// TIA Portal V19 export
FUNCTION_BLOCK "F_Zone29_FB"   // FB168, F_LAD
TITLE = SAFETY ZONE 29 - AREA 03 (SCARICO NAVETTA)
// stored: Access Published
   VAR
      D22_LightCurtain_Ext : "Door_FB";
      D24_LightCurtain_Int : "Door_FB";
      FNS : "ForceNormalStop";
      F_Sinamics_Navetta_Testa : "FDevice_Sinamics_FB";
      F_Sinamics_Navetta_Coda : "FDevice_Sinamics_FB";
      F_SafetyValve_Air_A0304 : "FDevice_Valve_FB";
   END_VAR
   VAR_TEMP
      DoorNormalStop : Bool;
      DoorSafeStop : Bool;
      Door_OK : Bool;
      FDBK : Bool;
   END_VAR
BEGIN

REGION Network 1: < < < < < < < < < < DOOR > > > > > > > > > >
END_REGION

REGION Network 2: Zone Entry enable
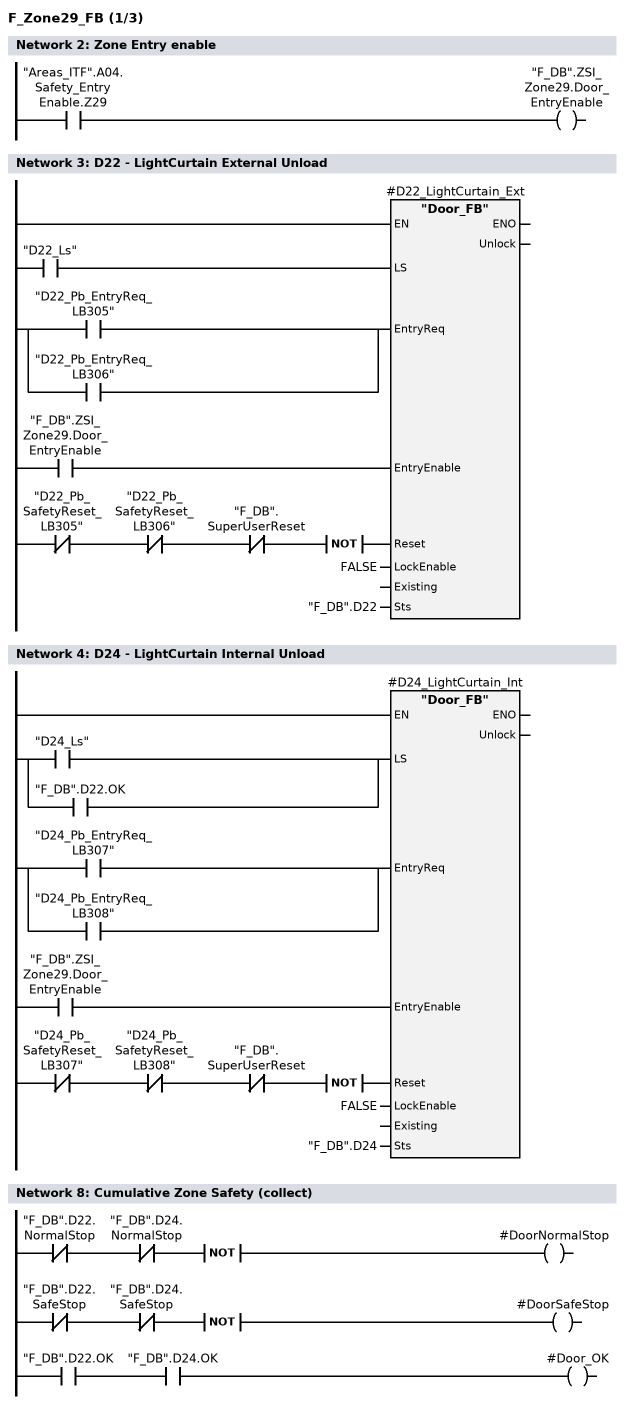
   RUNG wire#powerrail
      Contact( "Areas_ITF".A04.Safety_EntryEnable.Z29 )
      Coil( "F_DB".ZSI_Zone29.Door_EntryEnable )
   END_RUNG
   // the same network as SCL:
   "F_DB".ZSI_Zone29.Door_EntryEnable := "Areas_ITF".A04.Safety_EntryEnable.Z29;
END_REGION

REGION Network 3: D22 - LightCurtain External Unload
   RUNG wire#powerrail
      #D22_LightCurtain_Ext(LS := wire#w1, EntryReq := wire#w2, EntryEnable := wire#w3, Reset := wire#w4, LockEnable := FALSE, Existing :=, Sts := "F_DB".D22, Unlock =>)
   END_RUNG
   RUNG wire#powerrail
      Contact( "D22_Ls" )
   END_RUNG wire#w1
   RUNG wire#powerrail
      Contact( "D22_Pb_EntryReq_LB305" )
   END_RUNG wire#w2
   RUNG wire#powerrail
      Contact( "D22_Pb_EntryReq_LB306" )
   END_RUNG wire#w2
   RUNG wire#powerrail
      Contact( "F_DB".ZSI_Zone29.Door_EntryEnable )
   END_RUNG wire#w3
   RUNG wire#powerrail
      I_Contact( "D22_Pb_SafetyReset_LB305" )
      I_Contact( "D22_Pb_SafetyReset_LB306" )
      I_Contact( "F_DB".SuperUserReset )
      Not()
   END_RUNG wire#w4
   // the same network as SCL:
   #D22_LightCurtain_Ext(LS := "D22_Ls",   // "Door_FB"
                         EntryReq := "D22_Pb_EntryReq_LB305" OR "D22_Pb_EntryReq_LB306",
                         EntryEnable := "F_DB".ZSI_Zone29.Door_EntryEnable,
                         Reset := NOT (NOT "D22_Pb_SafetyReset_LB305" AND NOT "D22_Pb_SafetyReset_LB306" AND NOT "F_DB".SuperUserReset),
                         LockEnable := FALSE,
                         Sts := "F_DB".D22);
END_REGION

REGION Network 4: D24 - LightCurtain Internal Unload
   RUNG wire#powerrail
      #D24_LightCurtain_Int(LS := wire#w1, EntryReq := wire#w2, EntryEnable := wire#w3, Reset := wire#w4, LockEnable := FALSE, Existing :=, Sts := "F_DB".D24, Unlock =>)
   END_RUNG
   RUNG wire#powerrail
      Contact( "D24_Ls" )
   END_RUNG wire#w1
   RUNG wire#powerrail
      Contact( "F_DB".D22.OK )
   END_RUNG wire#w1
   RUNG wire#powerrail
      Contact( "D24_Pb_EntryReq_LB307" )
   END_RUNG wire#w2
   RUNG wire#powerrail
      Contact( "D24_Pb_EntryReq_LB308" )
   END_RUNG wire#w2
   RUNG wire#powerrail
      Contact( "F_DB".ZSI_Zone29.Door_EntryEnable )
   END_RUNG wire#w3
   RUNG wire#powerrail
      I_Contact( "D24_Pb_SafetyReset_LB307" )
      I_Contact( "D24_Pb_SafetyReset_LB308" )
      I_Contact( "F_DB".SuperUserReset )
      Not()
   END_RUNG wire#w4
   // the same network as SCL:
   #D24_LightCurtain_Int(LS := "D24_Ls" OR "F_DB".D22.OK,   // "Door_FB"
                         EntryReq := "D24_Pb_EntryReq_LB307" OR "D24_Pb_EntryReq_LB308",
                         EntryEnable := "F_DB".ZSI_Zone29.Door_EntryEnable,
                         Reset := NOT (NOT "D24_Pb_SafetyReset_LB307" AND NOT "D24_Pb_SafetyReset_LB308" AND NOT "F_DB".SuperUserReset),
                         LockEnable := FALSE,
                         Sts := "F_DB".D24);
END_REGION

REGION Network 7: < < < < < < < < < < ZONE SAFETY INTERFACE > > > > > > > > > >
END_REGION

REGION Network 8: Cumulative Zone Safety (collect)
   RUNG wire#powerrail
      I_Contact( "F_DB".D22.NormalStop )
      I_Contact( "F_DB".D24.NormalStop )
      Not()
      Coil( #DoorNormalStop )
   END_RUNG
   RUNG wire#powerrail
      I_Contact( "F_DB".D22.SafeStop )
      I_Contact( "F_DB".D24.SafeStop )
      Not()
      Coil( #DoorSafeStop )
   END_RUNG
   RUNG wire#powerrail
      Contact( "F_DB".D22.OK )
      Contact( "F_DB".D24.OK )
      Coil( #Door_OK )
   END_RUNG
   // the same network as SCL:
   #DoorNormalStop := NOT (NOT "F_DB".D22.NormalStop AND NOT "F_DB".D24.NormalStop);
   #DoorSafeStop := NOT (NOT "F_DB".D22.SafeStop AND NOT "F_DB".D24.SafeStop);
   #Door_OK := "F_DB".D22.OK AND "F_DB".D24.OK;
END_REGION

REGION Network 9: Zone must stay in Normal Stop During Restart
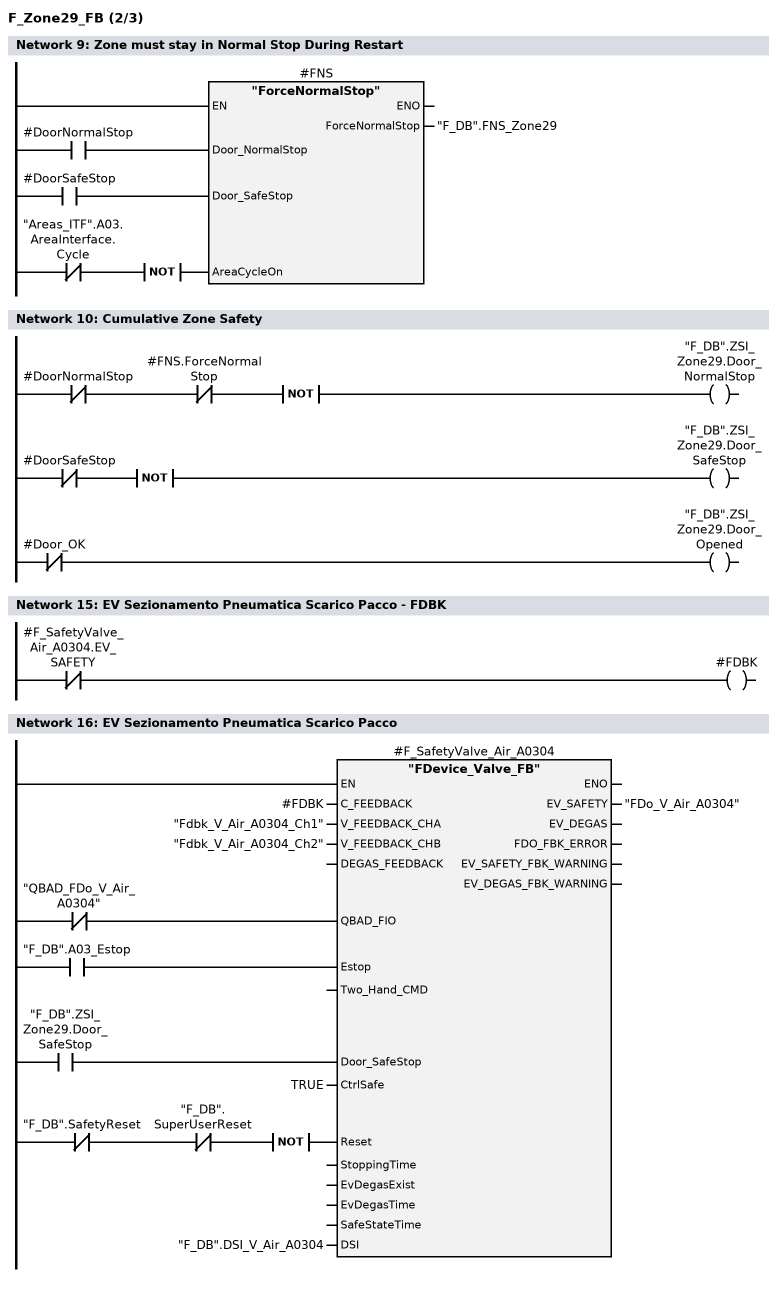
   RUNG wire#powerrail
      #FNS(Door_NormalStop := wire#w1, Door_SafeStop := wire#w2, AreaCycleOn := wire#w3, ForceNormalStop => "F_DB".FNS_Zone29)
   END_RUNG
   RUNG wire#powerrail
      Contact( #DoorNormalStop )
   END_RUNG wire#w1
   RUNG wire#powerrail
      Contact( #DoorSafeStop )
   END_RUNG wire#w2
   RUNG wire#powerrail
      I_Contact( "Areas_ITF".A03.AreaInterface.Cycle )
      Not()
   END_RUNG wire#w3
   // the same network as SCL:
   #FNS(Door_NormalStop := #DoorNormalStop,   // "ForceNormalStop"
        Door_SafeStop := #DoorSafeStop,
        AreaCycleOn := NOT (NOT "Areas_ITF".A03.AreaInterface.Cycle),
        ForceNormalStop => "F_DB".FNS_Zone29);
END_REGION

REGION Network 10: Cumulative Zone Safety
   RUNG wire#powerrail
      I_Contact( #DoorNormalStop )
      I_Contact( #FNS.ForceNormalStop )
      Not()
      Coil( "F_DB".ZSI_Zone29.Door_NormalStop )
   END_RUNG
   RUNG wire#powerrail
      I_Contact( #DoorSafeStop )
      Not()
      Coil( "F_DB".ZSI_Zone29.Door_SafeStop )
   END_RUNG
   RUNG wire#powerrail
      I_Contact( #Door_OK )
      Coil( "F_DB".ZSI_Zone29.Door_Opened )
   END_RUNG
   // the same network as SCL:
   "F_DB".ZSI_Zone29.Door_NormalStop := NOT (NOT #DoorNormalStop AND NOT #FNS.ForceNormalStop);
   "F_DB".ZSI_Zone29.Door_SafeStop := NOT (NOT #DoorSafeStop);
   "F_DB".ZSI_Zone29.Door_Opened := NOT #Door_OK;
END_REGION

REGION Network 11: >
END_REGION

REGION Network 12: >
END_REGION

REGION Network 13: < < < < < < < < < < DEVICES SAFETY VALVES > > > > > > > > > >
END_REGION

REGION Network 14: >
END_REGION

REGION Network 15: EV Sezionamento Pneumatica Scarico Pacco - FDBK
   RUNG wire#powerrail
      I_Contact( #F_SafetyValve_Air_A0304.EV_SAFETY )
      Coil( #FDBK )
   END_RUNG
   // the same network as SCL:
   #FDBK := NOT #F_SafetyValve_Air_A0304.EV_SAFETY;
END_REGION

REGION Network 16: EV Sezionamento Pneumatica Scarico Pacco
   RUNG wire#powerrail
      #F_SafetyValve_Air_A0304(QBAD_FIO := wire#w1, Estop := wire#w2, Door_SafeStop := wire#w3, Reset := wire#w4, C_FEEDBACK := #FDBK, V_FEEDBACK_CHA := "Fdbk_V_Air_A0304_Ch1", V_FEEDBACK_CHB := "Fdbk_V_Air_A0304_Ch2", DEGAS_FEEDBACK :=, Two_Hand_CMD :=, CtrlSafe := TRUE, StoppingTime :=, EvDegasExist :=, EvDegasTime :=, SafeStateTime :=, DSI := "F_DB".DSI_V_Air_A0304, EV_SAFETY => "FDo_V_Air_A0304", EV_DEGAS =>, FDO_FBK_ERROR =>, EV_SAFETY_FBK_WARNING =>, EV_DEGAS_FBK_WARNING =>)
   END_RUNG
   RUNG wire#powerrail
      I_Contact( "QBAD_FDo_V_Air_A0304" )
   END_RUNG wire#w1
   RUNG wire#powerrail
      Contact( "F_DB".A03_Estop )
   END_RUNG wire#w2
   RUNG wire#powerrail
      Contact( "F_DB".ZSI_Zone29.Door_SafeStop )
   END_RUNG wire#w3
   RUNG wire#powerrail
      I_Contact( "F_DB".SafetyReset )
      I_Contact( "F_DB".SuperUserReset )
      Not()
   END_RUNG wire#w4
   // the same network as SCL:
   #F_SafetyValve_Air_A0304(C_FEEDBACK := #FDBK,   // "FDevice_Valve_FB"
                           V_FEEDBACK_CHA := "Fdbk_V_Air_A0304_Ch1",
                           V_FEEDBACK_CHB := "Fdbk_V_Air_A0304_Ch2",
                           QBAD_FIO := NOT "QBAD_FDo_V_Air_A0304",
                           Estop := "F_DB".A03_Estop,
                           Door_SafeStop := "F_DB".ZSI_Zone29.Door_SafeStop,
                           CtrlSafe := TRUE,
                           Reset := NOT (NOT "F_DB".SafetyReset AND NOT "F_DB".SuperUserReset),
                           DSI := "F_DB".DSI_V_Air_A0304,
                           EV_SAFETY => "FDo_V_Air_A0304");
END_REGION

REGION Network 17: >
END_REGION

REGION Network 18: < < < < < < < < < < DEVICES CONTACTORS > > > > > > > > > >
END_REGION

REGION Network 19: >
END_REGION

REGION Network 20: >
END_REGION

REGION Network 21: < < < < < < < < < < DEVICES S120 > > > > > > > > > >
END_REGION

REGION Network 22: S120 - Ax Testa Navetta
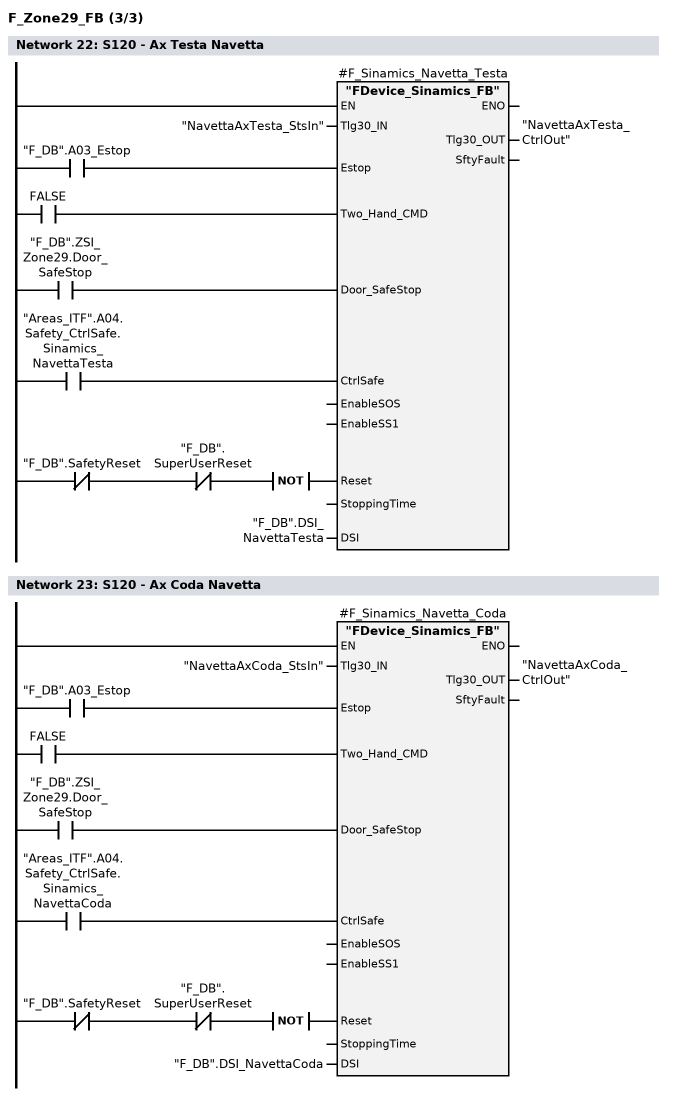
   RUNG wire#powerrail
      #F_Sinamics_Navetta_Testa(Estop := wire#w1, Two_Hand_CMD := wire#w2, Door_SafeStop := wire#w3, CtrlSafe := wire#w4, Reset := wire#w5, Tlg30_IN := "NavettaAxTesta_StsIn", EnableSOS :=, EnableSS1 :=, StoppingTime :=, DSI := "F_DB".DSI_NavettaTesta, Tlg30_OUT => "NavettaAxTesta_CtrlOut", SftyFault =>)
   END_RUNG
   RUNG wire#powerrail
      Contact( "F_DB".A03_Estop )
   END_RUNG wire#w1
   RUNG wire#powerrail
      Contact( FALSE )
   END_RUNG wire#w2
   RUNG wire#powerrail
      Contact( "F_DB".ZSI_Zone29.Door_SafeStop )
   END_RUNG wire#w3
   RUNG wire#powerrail
      Contact( "Areas_ITF".A04.Safety_CtrlSafe.Sinamics_NavettaTesta )
   END_RUNG wire#w4
   RUNG wire#powerrail
      I_Contact( "F_DB".SafetyReset )
      I_Contact( "F_DB".SuperUserReset )
      Not()
   END_RUNG wire#w5
   // the same network as SCL:
   #F_Sinamics_Navetta_Testa(Tlg30_IN := "NavettaAxTesta_StsIn",   // "FDevice_Sinamics_FB"
                           Estop := "F_DB".A03_Estop,
                           Two_Hand_CMD := FALSE,
                           Door_SafeStop := "F_DB".ZSI_Zone29.Door_SafeStop,
                           CtrlSafe := "Areas_ITF".A04.Safety_CtrlSafe.Sinamics_NavettaTesta,
                           Reset := NOT (NOT "F_DB".SafetyReset AND NOT "F_DB".SuperUserReset),
                           DSI := "F_DB".DSI_NavettaTesta,
                           Tlg30_OUT => "NavettaAxTesta_CtrlOut");
END_REGION

REGION Network 23: S120 - Ax Coda Navetta
   RUNG wire#powerrail
      #F_Sinamics_Navetta_Coda(Estop := wire#w1, Two_Hand_CMD := wire#w2, Door_SafeStop := wire#w3, CtrlSafe := wire#w4, Reset := wire#w5, Tlg30_IN := "NavettaAxCoda_StsIn", EnableSOS :=, EnableSS1 :=, StoppingTime :=, DSI := "F_DB".DSI_NavettaCoda, Tlg30_OUT => "NavettaAxCoda_CtrlOut", SftyFault =>)
   END_RUNG
   RUNG wire#powerrail
      Contact( "F_DB".A03_Estop )
   END_RUNG wire#w1
   RUNG wire#powerrail
      Contact( FALSE )
   END_RUNG wire#w2
   RUNG wire#powerrail
      Contact( "F_DB".ZSI_Zone29.Door_SafeStop )
   END_RUNG wire#w3
   RUNG wire#powerrail
      Contact( "Areas_ITF".A04.Safety_CtrlSafe.Sinamics_NavettaCoda )
   END_RUNG wire#w4
   RUNG wire#powerrail
      I_Contact( "F_DB".SafetyReset )
      I_Contact( "F_DB".SuperUserReset )
      Not()
   END_RUNG wire#w5
   // the same network as SCL:
   #F_Sinamics_Navetta_Coda(Tlg30_IN := "NavettaAxCoda_StsIn",   // "FDevice_Sinamics_FB"
                           Estop := "F_DB".A03_Estop,
                           Two_Hand_CMD := FALSE,
                           Door_SafeStop := "F_DB".ZSI_Zone29.Door_SafeStop,
                           CtrlSafe := "Areas_ITF".A04.Safety_CtrlSafe.Sinamics_NavettaCoda,
                           Reset := NOT (NOT "F_DB".SafetyReset AND NOT "F_DB".SuperUserReset),
                           DSI := "F_DB".DSI_NavettaCoda,
                           Tlg30_OUT => "NavettaAxCoda_CtrlOut");
END_REGION

REGION Network 24: >
END_REGION

REGION Network 25: >
END_REGION
END_FUNCTION_BLOCK
